TYPE st_Ledstrip_MachineData :
STRUCT
	r_SOC 					: REAL;
	r_DCCurrent				: REAL;
	e_systemStatus 			: eSystemStatus;
END_STRUCT
END_TYPE

(* stored: Version 1.1.0.1, ProductVersion 3.1.4026.18
   DUT st_Ledstrip_MachineData: Id {bd0f726c-c6d3-43da-a8ef-9fb161da9b4f} *)
